TYPE stAnalogueProcessData : 
STRUCT
    FailureDescription : STRING;
    Minimum : REAL;
    Maximum : REAL;
END_STRUCT
END_TYPE

(* stored: Version 1.1.0.1, ProductVersion 3.1.4024.6
   DUT stAnalogueProcessData: Id {4e8eaf20-b62b-4a8a-a572-e7b3b1744995} *)
